FUNCTION F_PressureSensorInToBar : LREAL
VAR_INPUT
	fPressure : LREAL;
END_VAR
VAR
END_VAR

F_PressureSensorInToBar := fPressure*400/32767;

END_FUNCTION

(* stored: Version 1.1.0.1, ProductVersion 3.1.4024.13
   POU F_PressureSensorInToBar: Id {ee464f70-e313-4580-902c-24224853dc35}, SpecialFunc None *)
